(* IEC 61131-3 sources: Sps24ProgettoDirectLoadingOOP/src/Libreria/OOP, 5 files *)

(* ---- UserDataType.st ---- *)
NAMESPACE libUdtOop

    TYPE
        gripperInterface : STRUCT
            gripperCmd : gripperCommands;
            gripperOpened : BOOL;
            gripperClosed : BOOL;
        END_STRUCT;
    END_TYPE

    TYPE
        gripperCommands : STRUCT
            openGripper : BOOL;
            closeGripper : BOOL;
        END_STRUCT;
    END_TYPE

    TYPE
        axisInterface : STRUCT
            axisCmd : axisCommands;
            axisOn : BOOL;
            axisReferenced : BOOL;
            axisError : BOOL;
            axisActualPosition : LREAL;
            axisPos1 : BOOL;
            axisPos2 : BOOL;
        END_STRUCT;
    END_TYPE

    TYPE
        axisCommands : STRUCT
            powerAxis : BOOL;
            homingAxis : BOOL;
            goToPos1Axis : BOOL;
            goToPos2Axis : BOOL;
        END_STRUCT;
    END_TYPE

    TYPE
        armInterface : STRUCT
            armCmd : armCommands;
            armPos1 : BOOL;
            armPos2 : BOOL;
            endPick : BOOL;
            endPlace : BOOL;
        END_STRUCT;
    END_TYPE

    TYPE
        armCommands : STRUCT
            pickArm : BOOL;
            placeArm : BOOL;
        END_STRUCT;
    END_TYPE

    TYPE
        POSITION : LREAL (
            NONE := 0,
            ARMPOS1 := 5.0,
            ARMPOS2 := 100.0,
            BUFFERPOS1 := 270.0,
            BUFFERPOS2 := 90.0,
            TOL := 0.5
        ) := NONE;
    END_TYPE
    TYPE
        DIRECTION : INT (
            DEFAULT := 3,
            STARTMODE := 1
        ) := DEFAULT;
    END_TYPE

    TYPE
        TIMER : LTIME (
            GRIPPER := LT#1s,
            WIP := LT#2s
        ) := GRIPPER;
    END_TYPE

END_NAMESPACE

(* ---- Arm.st ---- *)
USING libUdtOop;
USING Siemens.Simatic.S71500.MotionControl.Native;

NAMESPACE libMotOop

    CLASS PUBLIC ArmClass EXTENDS AxisClass
        VAR PUBLIC
            _instGripper : GripperClass;
            //_instAxis : AxisClass;
            _armInterface : armInterface;
        END_VAR

        METHOD PUBLIC Pick
            VAR
                state : INT;
            END_VAR
            //Logica Presa Braccio
            CASE state OF
                0: // Avvio Missione Prendi
                    IF _armInterface.armCmd.pickArm THEN
                        _armInterface.endPick := FALSE;
                        state := 2;
                    END_IF;
                2: // La pinza è aperta?
                    IF _instGripper._gripperInterface.gripperOpened THEN
                        state := 4;
                    ELSE
                        _instGripper.OpenGripper(timerGripper := TIMER#GRIPPER);
                    END_IF;
                4: //Vai a posizione di presa (bassa)
                    IF _armInterface.armPos1 THEN
                        state := 6;
                    ELSE
                        THIS.MoveAbs(direction := DIRECTION#DEFAULT, position := POSITION#ARMPOS1);
                    END_IF;
                6: //Chiudi la pinza
                    IF _instGripper._gripperInterface.gripperClosed THEN
                        state := 8;
                    ELSE
                        _instGripper.CloseGripper(timerGripper := TIMER#GRIPPER);
                    END_IF;
                8: //Vai a posizione di attesa (alta)
                    IF _armInterface.armPos2 THEN
                        state := 30;
                    ELSE
                        THIS.MoveAbs(direction := DIRECTION#DEFAULT, position := POSITION#ARMPOS2);
                    END_IF;
                30: //Fine
                    state := 0;
                    _armInterface.endPick := TRUE;
            END_CASE;
        END_METHOD

        METHOD PUBLIC Place
            VAR
                state : INT;
            END_VAR
            //Logica Posa Braccio
            CASE state OF
                0: // Avvio Missione Posa
                    IF _armInterface.armCmd.placeArm THEN
                        _armInterface.endPlace := FALSE;
                        state := 2;
                    END_IF;
                2: //Vai a posizione di posa (bassa)
                    IF _armInterface.armPos1 THEN
                        state := 4;
                    ELSE
                        THIS.MoveAbs(direction := DIRECTION#DEFAULT, position := POSITION#ARMPOS1);
                    END_IF;
                4: //Apri la pinza
                    IF _instGripper._gripperInterface.gripperOpened THEN
                        state := 6;
                    ELSE
                        _instGripper.OpenGripper(timerGripper := TIMER#GRIPPER);
                    END_IF;
                6: //Vai a posizione di attesa (alta)
                    IF _armInterface.armPos2 THEN
                        state := 30;
                    ELSE
                        THIS.MoveAbs(direction := DIRECTION#DEFAULT, position := POSITION#ARMPOS2);
                    END_IF;
                30: //Fine
                    state := 0;
                    _armInterface.endPlace := TRUE;
            END_CASE;
        END_METHOD
    END_CLASS

END_NAMESPACE

(* ---- Controller.st ---- *)
USING libUdtOop;
USING System.Timer;
USING Siemens.Simatic.S71500.MotionControl.Native;

NAMESPACE libMotOop

    FUNCTION_BLOCK controlloreCentrale
        VAR_INPUT
            start : BOOL;
            posAxisRot : DB_ANY;
            posAxisRight : DB_ANY;
            posAxisLeft : DB_ANY;
        END_VAR
        VAR_OUTPUT
            cicloAutomatico : BOOL;
        END_VAR
        VAR
            state : INT;
            timer : OnDelay;
            numeroCicli : INT;
            asseRot : AxisClass;
            asseDx : ArmClass;
            asseSx : ArmClass;
        END_VAR

        CASE state OF
            0: //one-time setup
                asseRot.SetAxis(posAxisRot);
                asseDx.SetAxis(posAxisRight);
                asseSx.SetAxis(posAxisLeft);
                state := 1;
            1: // Avvio Sequenza
                IF start THEN
                    state := 100;
                    cicloAutomatico := TRUE;
                    asseDx._armInterface.endPick := FALSE;
                    asseDx._armInterface.endPlace := FALSE;
                    asseSx._armInterface.endPick := FALSE;
                    asseSx._armInterface.endPlace := FALSE;
                END_IF;
            100: // Controllo se gli assi sono accesi
                IF asseRot._axisInterface.axisOn AND asseSx._axisInterface.axisOn AND asseDx._axisInterface.axisOn THEN
                    state := 101;
                ELSE
                    IF NOT asseRot._axisInterface.axisOn THEN
                        asseRot.Power(startMode := DIRECTION#STARTMODE);
                    END_IF;
                    IF NOT asseSx._axisInterface.axisOn THEN
                        asseSx.Power(startMode := DIRECTION#STARTMODE);
                    END_IF;
                    IF NOT asseDx._axisInterface.axisOn THEN
                        asseDx.Power(startMode := DIRECTION#STARTMODE);
                    END_IF;
                END_IF;
            101: //Controllo se gli assi sono referenziati
                IF asseRot._axisInterface.axisReferenced AND asseSx._axisInterface.axisReferenced AND asseDx._axisInterface.axisReferenced THEN
                    state := 2;
                ELSE
                    IF NOT asseRot._axisInterface.axisReferenced THEN
                        asseRot.Homing();
                    END_IF;
                    IF NOT asseSx._axisInterface.axisReferenced THEN
                        asseSx.Homing();
                    END_IF;
                    IF NOT asseDx._axisInterface.axisReferenced THEN
                        asseDx.Homing();
                    END_IF;
                END_IF;
            2: // Ruota AsseRot in Pos 1
                IF asseRot._axisInterface.axisPos1 THEN
                    state := 4;
                ELSE
                    asseRot.MoveAbs(direction := DIRECTION#DEFAULT, position := POSITION#BUFFERPOS1);
                END_IF;
            4: // Prendi con AsseSx
                IF asseSx._armInterface.endPick THEN
                    asseSx._armInterface.endPick := FALSE;
                    state := 6;
                ELSE
                    asseSx.Pick();
                END_IF;
            6: // Attesa
                timer(signal := TRUE, duration := TIMER#WIP);
                IF timer.output THEN
                    timer.signal := FALSE;
                    state := 8;
                END_IF;
            8: // Posa con AsseSx
                IF asseSx._armInterface.endPlace THEN
                    asseSx._armInterface.endPlace := FALSE;
                    state := 10;
                ELSE
                    asseSx.Place();
                END_IF;
            10: // Ruota AsseRot in Pos 2
                IF asseRot._axisInterface.axisPos2 THEN
                    state := 12;
                ELSE
                    asseRot.MoveAbs(direction := DIRECTION#DEFAULT, position := POSITION#BUFFERPOS2);
                END_IF;
            12: // Prendi con AsseDx
                IF asseDx._armInterface.endPick THEN
                    asseDx._armInterface.endPick := FALSE;
                    state := 14;
                ELSE
                    asseDx.Pick();
                END_IF;
            14: //Attesa
                timer(signal := TRUE, duration := TIMER#WIP);
                IF timer.output THEN
                    timer.signal := FALSE;
                    state := 16;
                END_IF;
            16: // Posa con AsseDx
                IF asseDx._armInterface.endPlace THEN
                    asseDx._armInterface.endPlace := FALSE;
                    state := 30;
                ELSE
                    asseDx.Place();
                END_IF;
            30: //Fine Sequenza
                state := 1;
                cicloAutomatico := FALSE;
                numeroCicli := numeroCicli + 1;
        END_CASE;

        asseRot.CyclicCall();
        asseRot.CalculatePosition(POSITION#BUFFERPOS1, POSITION#BUFFERPOS2);

        asseDx.CyclicCall();
        asseDx.CalculatePosition(POSITION#ARMPOS1, POSITION#ARMPOS2);

        asseSx.CyclicCall();
        asseSx.CalculatePosition(POSITION#ARMPOS1, POSITION#ARMPOS2);

    END_FUNCTION_BLOCK

END_NAMESPACE

(* ---- Gripper.st ---- *)
USING libUdtOop;
USING System.Timer;

NAMESPACE libMotOop

    CLASS PUBLIC GripperClass
        VAR PROTECTED
            _instTimerOpen : OnDelay;
            _instTimerClose : OnDelay;
        END_VAR
        VAR PUBLIC
            _gripperInterface : gripperInterface;
        END_VAR

        METHOD PUBLIC OpenGripper
            VAR_INPUT
                timerGripper : LTIME;
            END_VAR
            _gripperInterface.gripperCmd.openGripper := TRUE;
            _instTimerOpen(signal := TRUE, duration := timerGripper, output => _gripperInterface.gripperOpened);
        END_METHOD

        METHOD PUBLIC CloseGripper
            VAR_INPUT
                timerGripper : LTIME;
            END_VAR
            _gripperInterface.gripperCmd.closeGripper := TRUE;
            _instTimerClose(signal := TRUE, duration := timerGripper, output => _gripperInterface.gripperClosed);
        END_METHOD
    END_CLASS

END_NAMESPACE

(* ---- program2.st ---- *)
USING libMotOop;
USING libUdtOop;
USING Siemens.Simatic.S71500.MotionControl.Native;

PROGRAM MyProgram2
    VAR_EXTERNAL
        start : BOOL;
        tavolaRotante : axisInterface;
        braccioDx : axisInterface;
        braccioSx : axisInterface;
        fineCiclo : BOOL;
    END_VAR

    VAR
        instControllore : controlloreCentrale;
    END_VAR

    VAR CONSTANT
        posAxisLeftDB  : UINT := UINT#3;
        posAxisRightDB  : UINT := UINT#6;
        posAxisRotDB  : UINT := UINT#16;
    END_VAR

    VAR_TEMP
        //posAxisLeftDBRef  : REF_TO TO_PositioningAxis;
        //posAxisRightDBRef  : REF_TO TO_PositioningAxis;
        //posAxisRotDBRef  : REF_TO TO_PositioningAxis;
    END_VAR

    //posAxisRotDBRef := AsPositioningAxisRef(posAxisRotDB);
    //posAxisLeftDBRef := AsPositioningAxisRef(posAxisLeftDB);
    //posAxisRightDBRef := AsPositioningAxisRef(posAxisRightDB);

    instControllore(start := start, posAxisRot := posAxisRotDB, posAxisRight := posAxisRightDB, posAxisLeft := posAxisLeftDB, cicloAutomatico => fineCiclo);

END_PROGRAM
